PROGRAM TESTER_C8
VAR
	TMR11: TON;
	TMR12: TON;
	TMR10: TON;
	TMR8: TON;
	TMR9: TON;
	TMR7: TON;
	TMR3: TON;
	TP1: TP;
	TMR1: TON;
	START_ROBOT: TP;
	TP2: TP;
	O_G6_HANG: BOOL;
	I_G6_HANG: BOOL;
	TMR2: TON;
	GO_ROBOT: BOOL;
	TP3: TP;
	TMR4: TON;
	CNT_CYCLE: CTU;
	START_ROTATE: R_TRIG;
	IN: INT;
	TMR_RELEASE: TON;
	TMR_OFF_MCAL: TON;
	TMR_RLS_SCAN: TON;
	AFTER_SCAN: BOOL;

	AFTER_SCAN1: BOOL;
	TMR_RLS_SCAN1: TON;
	C8_SEQ: INT;
	DLY1: TON;
	DLY2: TON;
	TMR_RLS: TON;
	TMR_RST: TON;
END_VAR


//GRIPPING CONTROL
IF TESTER_C8_VAR.I_C8_GRIPPER THEN
		TESTER_C8_VAR.O_C8_GRIPPER_CLOSE:=TRUE;
		TESTER_C8_VAR.O_C8_GRIPPER_OPEN:=FALSE;
ELSE
		TESTER_C8_VAR.O_C8_GRIPPER_CLOSE:=FALSE;
		TESTER_C8_VAR.O_C8_GRIPPER_OPEN:=TRUE;
END_IF

IF TESTER_C8_VAR.I_C8_SERROR THEN
	POWER_CONTROL.O_PWR_CTRL_ROBOT_C8:=TRUE;
	TMR_RELEASE(IN:=TRUE,PT:=T#0.5S);
	IF TMR_RELEASE.Q THEN
		POWER_CONTROL.O_PWR_CTRL_ROBOT_C8:=FALSE;
	END_IF
ELSE
	TMR_RELEASE(IN:=FALSE);	
END_IF

//MCAL
	IF TESTER_C8_VAR.I_C8_MCAL_REQUEST THEN
		TESTER_C8_VAR.O_G6_SELROBOT_2:=TRUE;
		IF TESTER_C8_VAR.O_G6_SELROBOT_2 THEN
			DLY1(IN:=TRUE,PT:=T#1S);
			IF DLY1.Q THEN
				TESTER_C8_VAR.O_G6_SETMOTORON:=TRUE;
			END_IF
			IF TESTER_C8_VAR.I_C8_MOTORON THEN
				DLY2(IN:=TRUE,PT:=T#1S);
				IF DLY2.Q THEN
					TESTER_C8_VAR.O_G6_MCAL:=TRUE;
					TMR_OFF_MCAL(IN:=TRUE,PT:=T#2S);	
				END_IF
				IF TMR_OFF_MCAL.Q THEN
					//TESTER_C8_VAR.O_G6_SELROBOT_2:=FALSE;
					//TESTER_C8_VAR.O_G6_MCAL:=FALSE;
				END_IF
			END_IF
		END_IF
	ELSE
		TESTER_C8_VAR.O_G6_SELROBOT_2:=FALSE;
		TESTER_C8_VAR.O_G6_MCAL:=FALSE;
		TMR_OFF_MCAL(IN:=FALSE);
		DLY1(IN:=FALSE);
		DLY2(IN:=FALSE);
	END_IF
	
IF NOT TESTER_C8_VAR.I_C8_MCAL_REQUEST AND TESTER_C8_VAR.C8_ERROR_1 >0 OR (TESTER_C8_VAR.C8_ERROR_2 >0 AND TESTER_C8_VAR.C8_ERROR_2 <32) OR TESTER_C8_VAR.I_C8_ERROR THEN
	TESTER_C8_VAR.O_G6_STOP:=TRUE;
	TMR_RST(IN:=TESTER_C8_VAR.O_G6_STOP,PT:=T#1S);
	IF TMR_RST.Q AND TESTER_C8_VAR.I_C8_READY THEN
		TESTER_C8_VAR.O_G6_STOP:=FALSE;
		TESTER_C8_VAR.O_G6_RESET:=TRUE;
		TMR_RST(IN:=FALSE);
	END_IF
ELSE
	TESTER_C8_VAR.O_G6_RESET:=FALSE;
	IF NOT TESTER_C8_VAR.I_C8_MOTORON THEN
		IF TESTER_C8_VAR.I_C8_READY AND NOT TESTER_C8_VAR.I_C8_ESTOPON AND NOT TESTER_C8_VAR.I_C8_SAFEGUARDON THEN
			TESTER_C8_VAR.O_G6_SETMOTORON:=TRUE;
			TESTER_C8_VAR.O_G6_SETMOTOROFF:=FALSE;	
		END_IF
	ELSE
		TESTER_C8_VAR.O_G6_SETMOTORON:=FALSE;
		TESTER_C8_VAR.O_G6_SETMOTOROFF:=FALSE;
	END_IF 
	IF TESTER_C8_VAR.O_C8_ENABLE AND NOT TESTER_C8_VAR.O_G6_MCAL THEN
		//TESTER_C8_VAR.O_G6_SELROBOT_2:=FALSE;
		IF NOT TESTER_C8_VAR.I_C8_ESTOPON AND NOT TESTER_C8_VAR.I_C8_SAFEGUARDON AND TESTER_C8_VAR.I_C8_READY THEN
			TESTER_C8_VAR.O_G6_SETMOTORON:=TRUE;
			TESTER_C8_VAR.O_G6_SETMOTOROFF:=FALSE;
		END_IF
		

		IF FLAG_VAR.ALLOW_EXECUTE_C8 AND NOT TESTER_C8_VAR.C8_ONDUTY THEN
			TESTER_C8_VAR.C8_START_MOVING:=TRUE;
			IF TESTER_C8_VAR.I_C8_RUNNING THEN
				TESTER_C8_VAR.O_G6_CONTINUE:=TRUE;
			END_IF
			IF TESTER_C8_VAR.I_C8_READY THEN
				TESTER_C8_VAR.O_G6_START:=TRUE;
			END_IF	 
			C8_SEQ:=1;
			ELSE
			TESTER_C8_VAR.O_G6_CONTINUE:=FALSE;
		END_IF
//EXECUTE MOVEMENT	
		IF TESTER_C8_VAR.I_C8_MOTORON AND  TESTER_C8_VAR.C8_START_MOVING AND NOT TESTER_C8_VAR.I_C8_ERROR THEN

			IF TESTER_C8_VAR.I_C8_ROTATE_INDEXING_2  AND NOT LOADER_VAR.I_CARRIER_DETECT_2 THEN
				TESTER_C8_VAR.READY_INDEXING:=TRUE;	
			END_IF
		
			CASE  C8_SEQ OF	
			1:
				FLAG_VAR.ALLOW_EXECUTE_C8:=FALSE;
				TESTER_C8_VAR.C8_MOVEMENT_SOURCE:=TESTER_C8_VAR.C8_MACHINE_POSITION.SOURCE_COORDINATE;
				TESTER_C8_VAR.C8_MOVEMENT_DESTINATION:=TESTER_C8_VAR.C8_MACHINE_POSITION.DESTINATION_COORDINATE;
				C8_SEQ:=2;
				TESTER_C8_VAR.O_G6_FINISH_SCANBARCODE :=FALSE;
			2:
//MOVEMENT TYPE
				IF NOT TESTER_C8_VAR.C8_ONDUTY THEN
					IF TESTER_C8_VAR.C8_MACHINE_POSITION.SOURCE_COORDINATE=0 AND TESTER_C8_VAR.C8_MACHINE_POSITION.DESTINATION_COORDINATE >0 THEN
						TESTER_C8_VAR.C8_PUTON:=TRUE;
						TESTER_C8_VAR.C8_TAKING:=FALSE;
						TESTER_C8_VAR.C8_TRANSFER:=FALSE;
						C8_SEQ:=3;
					END_IF
					 IF TESTER_C8_VAR.C8_MACHINE_POSITION.SOURCE_COORDINATE>0 AND TESTER_C8_VAR.C8_MACHINE_POSITION.DESTINATION_COORDINATE =0 THEN
						TESTER_C8_VAR.C8_PUTON:=FALSE;
						TESTER_C8_VAR.C8_TAKING:=TRUE;
						TESTER_C8_VAR.C8_TRANSFER:=FALSE;
						C8_SEQ:=3;
					END_IF
				 	IF TESTER_C8_VAR.C8_MACHINE_POSITION.SOURCE_COORDINATE>0 AND TESTER_C8_VAR.C8_MACHINE_POSITION.DESTINATION_COORDINATE >0 THEN
						TESTER_C8_VAR.C8_PUTON:=FALSE;
						TESTER_C8_VAR.C8_TAKING:=FALSE;
						TESTER_C8_VAR.C8_TRANSFER:=TRUE;
						C8_SEQ:=3;
					END_IF
				END_IF
3:
//ON DUTY CONTROL
			IF TESTER_C8_VAR.C8_PUTON OR TESTER_C8_VAR.C8_TAKING OR TESTER_C8_VAR.C8_TRANSFER AND NOT TESTER_C8_VAR.I_C8_FREE THEN
				TESTER_C8_VAR.C8_ONDUTY :=TRUE;
			ELSE
				TESTER_C8_VAR.C8_ONDUTY :=FALSE;
			END_IF
//MOVE CARRIER JIG FROM INDEXING TO MACHINE
			IF TESTER_C8_VAR.C8_PUTON THEN
				IF TESTER_C8_VAR.I_C8_READY THEN
					TESTER_C8_VAR.O_G6_START :=TRUE;
					TESTER_C8_VAR.O_G6_CONTINUE :=FALSE;
				ELSE
					TESTER_C8_VAR.O_G6_START :=FALSE;
				END_IF
				
				(*IF TESTER_C8_VAR.I_C8_READY_SCAN THEN
					TESTER_C8_VAR.O_G6_FINISH_SCANBARCODE :=TRUE;
					AFTER_SCAN:=TRUE ;
				END_IF*)
				//TESTER_C8_VAR.O_G6_FINISH_SCANBARCODE :=TESTER_C8_VAR.I_C8_READY_SCAN;
				IF TESTER_C8_VAR.O_G6_FINISH_SCANBARCODE THEN
					AFTER_SCAN:=TRUE;
				END_IF
				IF TESTER_C8_VAR.I_C8_RUNNING  AND NOT AFTER_SCAN AND NOT TESTER_C8_VAR.I_C8_FREE THEN
					TESTER_C8_VAR.O_G6_START :=FALSE;
				//	TESTER_C8_VAR.O_G6_CONTINUE :=TRUE;
				END_IF
				
				TMR_RLS_SCAN(IN:=AFTER_SCAN,PT:=T#1S);
				IF TMR_RLS_SCAN.Q THEN
						TESTER_C8_VAR.O_G6_FINISH_SCANBARCODE :=FALSE;
						TESTER_C8_VAR.O_G6_CONTINUE :=FALSE;
						TESTER_C8_VAR.C8_PUTON:=FALSE;
						AFTER_SCAN:=FALSE;
						TMR_RLS_SCAN(IN:=FALSE);
						C8_SEQ:=4;
						
				END_IF
			END_IF
//RETURN CARRIER JIG TO INDEXING				
			IF TESTER_C8_VAR.C8_TAKING THEN
				IF TESTER_C8_VAR.I_C8_RUNNING  AND NOT AFTER_SCAN1 THEN
					TESTER_C8_VAR.O_G6_START :=FALSE;
					TESTER_C8_VAR.O_G6_CONTINUE :=TRUE;
				END_IF
				(*IF TESTER_C8_VAR.I_C8_READY_SCAN THEN
					TESTER_C8_VAR.O_G6_FINISH_SCANBARCODE :=TRUE;
					AFTER_SCAN1:=TRUE;
				END_IF*)
				//TESTER_C8_VAR.O_G6_FINISH_SCANBARCODE :=TESTER_C8_VAR.I_C8_READY_SCAN;
				IF TESTER_C8_VAR.O_G6_FINISH_SCANBARCODE THEN
					AFTER_SCAN1:=TRUE;
				END_IF
				TMR_RLS_SCAN1(IN:=AFTER_SCAN1,PT:=T#1S);
				IF TMR_RLS_SCAN1.Q THEN
						TESTER_C8_VAR.O_G6_FINISH_SCANBARCODE :=FALSE;
						TESTER_C8_VAR.O_G6_CONTINUE :=FALSE;
						TESTER_C8_VAR.C8_TAKING:=FALSE;
						AFTER_SCAN1:=FALSE;
						TMR_RLS_SCAN1(IN:=FALSE);
						C8_SEQ:=4;
				END_IF
			END_IF
4:		
		IF TESTER_C8_VAR.I_C8_FREE THEN
			TESTER_C8_VAR.C8_START_MOVING:=FALSE;
			TESTER_C8_VAR.C8_ONDUTY:=FALSE;
			FLAG_VAR.ALLOW_EXECUTE_C8:=FALSE;
			TESTER_C8_VAR.O_G6_CONTINUE:=FALSE;
			TESTER_C8_VAR.O_G6_FINISH_SCANBARCODE :=FALSE;
			C8_SEQ:=0;
		ELSE
			TESTER_C8_VAR.O_G6_FINISH_SCANBARCODE :=TRUE;
		END_IF
END_CASE	
//AUTO RESET CONTINUE	
TMR_RLS(IN:=TESTER_C8_VAR.O_G6_CONTINUE,PT:=T#1S);
IF TMR_RLS.Q THEN
	TESTER_C8_VAR.O_G6_CONTINUE:=FALSE;
	TMR_RLS(IN:=FALSE);
END_IF
END_IF		
	ELSE
		IF NOT TESTER_C8_VAR.O_G6_MCAL THEN
			TESTER_C8_VAR.O_G6_SETMOTORON:=FALSE;
			TESTER_C8_VAR.O_G6_SETMOTOROFF:=TRUE;
			TESTER_C8_VAR.O_G6_SELROBOT_2:=FALSE;
		END_IF
	END_IF
END_IF

END_PROGRAM

(* stored: Version 1.1.0.1, ProductVersion 3.1.4020.12
   POU TESTER_C8: Id {0dcdbe04-b593-4d16-b09a-c3568efe4317}, SpecialFunc None *)
